Staubli VAL3: testAssembly.dtx

public dio dDio_Sucker = {link=valve1}
public dio dDio_Gripper = {link=valve2}
public tool tTool_3 = {z=179.5, fatherId=flange[0], ioLink=valve2}
public tool tTool_1 = {y=56.52, z=186.17, fatherId=flange[0], ioLink=valve1}
public tool tTool_2 = {y=100, z=136, fatherId=flange[0], ioLink=valve1}
mdesc mNomSpeed
public mdesc mMdesc_Move = {accel=50, vel=50, decel=50, tmax=50000, rmax=50000, leave=25, reach=25}
public mdesc mMdesc_Approach = {accel=20, vel=20, decel=20, tmax=20000, rmax=20000, leave=10, reach=10}
public mdesc mMdesc_Assembly = {accel=10, vel=10, decel=10, tmax=9999, rmax=9999, leave=5, reach=5}
public pointRx pPointRx_Task1[11]
  [0] = {fatherId=world[0]}
  [1] = {x=470.553007, y=-36.92597, z=-100.00047708, rx=-0.00159897, ry=179.996228, rz=0.00184176, fatherId=world[0]}
  [2] = {x=462.557886, y=-40.775959, z=-370.000522428, rx=-0.00112655, ry=179.996342, rz=0.0015039, fatherId=world[0]}
  [3] = {x=462.557886, y=-40.775959, z=-384.955213, rx=-0.00112655, ry=179.996342, rz=0.0015039, fatherId=world[0]}
  [4] = {x=462.557886, y=-40.775959, z=-370.000522428, rx=-0.00112655, ry=179.996342, rz=0.0015039, fatherId=world[0]}
  [5] = {x=462.559535, y=-40.775006, z=-100.00282324, rx=-0.00122429, ry=179.994784, rz=0.00157067, fatherId=world[0]}
  [6] = {x=758.545046, y=166.813373, z=-100.00327697, rx=-0.000742721, ry=179.994769, rz=0.00146888, fatherId=world[0]}
  [7] = {x=755.514304, y=158.963123, z=-333.864783, rx=-0.00147681, ry=179.996751, rz=0.00159201, fatherId=world[0]}
  [8] = {x=755.969382, y=158.33069, z=-366.778404, rx=-0.0014733, ry=179.996625, rz=0.00163886, fatherId=world[0]}
  [9] = {x=755.514304, y=158.963123, z=-333.864783, rx=-0.00147681, ry=179.996751, rz=0.00159201, fatherId=world[0]}
  [10] = {x=755.969382, y=158.33069, z=-100.000545775, rx=-0.00128229, ry=179.995583, rz=0.00173611, fatherId=world[0]}
public pointRx pPointRx_Task2[79]
  [0] = {fatherId=world[0]}
  [1] = {x=784.49936, y=235.445502, z=-49.999237, rx=-2.0204801, ry=113.232882, rz=-88.159509, fatherId=world[0]}
  [2] = {x=786.480486, y=262.552374, z=-299.99927, rx=-2.021757, ry=113.233517, rz=-88.158554, fatherId=world[0]}
  [3] = {x=784.36757, y=256.364439, z=-345.556165, rx=-2.0209842, ry=113.233476, rz=-88.159084, fatherId=world[0]}
  [4] = {x=784.367581, y=247.925511, z=-345.556163, rx=-2.0231337, ry=113.233887, rz=-88.157391, fatherId=world[0]}
  [5] = {x=784.367567, y=246.0220172, z=-341.350417, rx=-2.0233352, ry=113.233862, rz=-88.157219, fatherId=world[0]}
  [6] = {x=784.367581, y=242.656369, z=-336.237706, rx=-2.023434, ry=113.233818, rz=-88.157128, fatherId=world[0]}
  [7] = {x=784.367581, y=237.905853, z=-330.769653, rx=-2.023356, ry=113.233757, rz=-88.15718, fatherId=world[0]}
  [8] = {x=784.367581, y=232.925388, z=-325.864693, rx=-2.0234471, ry=113.233755, rz=-88.157103, fatherId=world[0]}
  [9] = {x=784.367581, y=228.681059, z=-321.473257, rx=-2.0234581, ry=113.233761, rz=-88.157095, fatherId=world[0]}
  [10] = {x=784.36758, y=224.624968, z=-318.39244, rx=-2.023448, ry=113.233762, rz=-88.157103, fatherId=world[0]}
  [11] = {x=784.367571, y=220.157122, z=-315.888328, rx=-2.0231771, ry=113.233735, rz=-88.157321, fatherId=world[0]}
  [12] = {x=784.36758, y=215.623373, z=-312.784136, rx=-2.0234496, ry=113.233801, rz=-88.157109, fatherId=world[0]}
  [13] = {x=784.367578, y=187.857141, z=-309.784137, rx=-2.0235808, ry=113.233878, rz=-88.157017, fatherId=world[0]}
  [14] = {x=784.368404, y=149.380411, z=-325.728255, rx=-2.0259223, ry=113.23421, rz=-88.155082, fatherId=world[0]}
  [15] = {x=784.36842, y=116.303705, z=-343.9057, rx=-2.0259843, ry=113.234309, rz=-88.155037, fatherId=world[0]}
  [16] = {x=786.563391, y=116.321118, z=-358.0200991, rx=-2.0241413, ry=113.234116, rz=-88.156874, fatherId=world[0]}
  [17] = {x=786.563381, y=124.191183, z=-358.108912, rx=-2.0225404, ry=113.233983, rz=-88.158152, fatherId=world[0]}
  [18] = {x=786.563391, y=124.767216, z=-356.140228, rx=-2.0223811, ry=113.233934, rz=-88.158276, fatherId=world[0]}
  [19] = {x=786.563381, y=126.602377, z=-350.283386, rx=-2.0218675, ry=113.233782, rz=-88.158676, fatherId=world[0]}
  [20] = {x=786.563381, y=128.973279, z=-344.998769, rx=-2.021688, ry=113.233689, rz=-88.158812, fatherId=world[0]}
  [21] = {x=786.563381, y=130.903655, z=-341.475635, rx=-2.0216225, ry=113.233645, rz=-88.158861, fatherId=world[0]}
  [22] = {x=786.56339, y=133.536756, z=-336.64486, rx=-2.0217804, ry=113.233636, rz=-88.158733, fatherId=world[0]}
  [23] = {x=786.563381, y=136.419075, z=-333.330297, rx=-2.0221318, ry=113.233692, rz=-88.158455, fatherId=world[0]}
  [24] = {x=786.56338, y=139.330018, z=-329.891057, rx=-2.021782, ry=113.233625, rz=-88.158731, fatherId=world[0]}
  [25] = {x=786.56338, y=143.199956, z=-325.866072, rx=-2.0218296, ry=113.233633, rz=-88.158694, fatherId=world[0]}
  [26] = {x=786.56338, y=146.30778, z=-323.413807, rx=-2.0218444, ry=113.23365, rz=-88.158684, fatherId=world[0]}
  [27] = {x=786.56338, y=149.408417, z=-321.184959, rx=-2.0221042, ry=113.233703, rz=-88.15848, fatherId=world[0]}
  [28] = {x=786.56338, y=154.738391, z=-317.954673, rx=-2.0217603, ry=113.233663, rz=-88.158754, fatherId=world[0]}
  [29] = {x=786.563389, y=158.0830096, z=-315.867788, rx=-2.0216758, ry=113.233652, rz=-88.158821, fatherId=world[0]}
  [30] = {x=786.563379, y=164.0860287, z=-313.649177, rx=-2.0215778, ry=113.233658, rz=-88.158902, fatherId=world[0]}
  [31] = {x=786.563379, y=170.136337, z=-312.205266, rx=-2.0219197, ry=113.233709, rz=-88.158631, fatherId=world[0]}
  [32] = {x=786.563377, y=202.68066, z=-312.205267, rx=-2.0217657, ry=113.233694, rz=-88.158755, fatherId=world[0]}
  [33] = {x=786.562888, y=216.0691273, z=-300.938154, rx=-2.0195136, ry=113.233344, rz=-88.160612, fatherId=world[0]}
  [34] = {x=786.562876, y=231.0113823, z=-300.938159, rx=-2.0171914, ry=113.232942, rz=-88.162452, fatherId=world[0]}
  [35] = {x=786.563361, y=231.0085614, z=-320.286213, rx=-2.0186299, ry=113.233599, rz=-88.161422, fatherId=world[0]}
  [36] = {x=784.474315, y=225.309214, z=-319.0657028, rx=-1.651499, ry=118.747777, rz=-88.567983, fatherId=world[0]}
  [37] = {x=784.474296, y=222.251329, z=-316.987746, rx=-1.652221, ry=118.747936, rz=-88.567442, fatherId=world[0]}
  [38] = {x=784.474315, y=217.578441, z=-314.772279, rx=-1.653461, ry=118.748225, rz=-88.566518, fatherId=world[0]}
  [39] = {x=784.474315, y=215.091758, z=-313.46553, rx=-1.654105, ry=118.748369, rz=-88.566037, fatherId=world[0]}
  [40] = {x=784.474314, y=206.499598, z=-313.465531, rx=-1.654999, ry=118.748116, rz=-88.565412, fatherId=world[0]}
  [41] = {x=784.474089, y=192.932163, z=-313.465215, rx=-1.654882, ry=118.747943, rz=-88.565623, fatherId=world[0]}
  [42] = {x=784.474673, y=178.17243, z=-313.464776, rx=-1.656821, ry=118.748298, rz=-88.564166, fatherId=world[0]}
  [43] = {x=784.474672, y=174.260972, z=-313.464777, rx=-1.656939, ry=118.748314, rz=-88.564078, fatherId=world[0]}
  [44] = {x=784.475657, y=168.377273, z=-315.634673, rx=-1.658494, ry=118.748564, rz=-88.563064, fatherId=world[0]}
  [45] = {x=784.475669, y=164.260614, z=-317.844146, rx=-1.658331, ry=118.748528, rz=-88.563185, fatherId=world[0]}
  [46] = {x=784.475656, y=160.796344, z=-320.542356, rx=-1.658243, ry=118.748527, rz=-88.563255, fatherId=world[0]}
  [47] = {x=784.475656, y=158.320085, z=-323.932867, rx=-1.6584, ry=118.74857, rz=-88.56314, fatherId=world[0]}
  [48] = {x=784.975647, y=155.528626, z=-326.455306, rx=-1.658273, ry=118.748538, rz=-88.563234, fatherId=world[0]}
  [49] = {x=784.976148, y=153.315191, z=-328.0961238, rx=-1.598646, ry=119.905815, rz=-88.631144, fatherId=world[0]}
  [50] = {x=785.626772, y=149.240023, z=-328.814604, rx=-1.599447, ry=120.005925, rz=-88.630678, fatherId=world[0]}
  [51] = {x=786.767462, y=147.46738, z=-331.0758995, rx=-1.60019, ry=120.205812, rz=-88.629945, fatherId=world[0]}
  [52] = {x=787.815814, y=145.632313, z=-333.126809, rx=-1.600796, ry=120.405903, rz=-88.629498, fatherId=world[0]}
  [53] = {x=789.569891, y=142.636972, z=-335.419631, rx=-1.601401, ry=120.555967, rz=-88.629047, fatherId=world[0]}
  [54] = {x=790.459284, y=141.85958, z=-337.809684, rx=-1.559394, ry=120.763388, rz=-88.67702, fatherId=world[0]}
  [55] = {x=791.982542, y=140.32981, z=-341.122996, rx=-1.544512, ry=121.0929413, rz=-88.694365, fatherId=world[0]}
  [56] = {x=792.275209, y=138.662447, z=-342.192906, rx=-1.519234, ry=121.653145, rz=-88.723629, fatherId=world[0]}
  [57] = {x=792.536625, y=138.572731, z=-345.0027193, rx=-1.519371, ry=121.653161, rz=-88.72353, fatherId=world[0]}
  [58] = {x=793.732094, y=138.572712, z=-347.743766, rx=-1.519449, ry=121.653157, rz=-88.723472, fatherId=world[0]}
  [59] = {x=794.288171, y=138.57273, z=-351.481062, rx=-1.519558, ry=121.653153, rz=-88.723392, fatherId=world[0]}
  [60] = {x=795.749739, y=138.572695, z=-352.856774, rx=-1.464073, ry=122.955659, rz=-88.788175, fatherId=world[0]}
  [61] = {x=794.971485, y=136.0698573, z=-356.118195, rx=-1.465483, ry=122.955943, rz=-88.787448, fatherId=world[0]}
  [62] = {x=794.0815342, y=136.0693946, z=-359.869106, rx=-1.418998, ry=124.145823, rz=-88.84234, fatherId=world[0]}
  [63] = {x=793.373601, y=136.0693624, z=-361.302488, rx=-1.441168, ry=123.608884, rz=-88.816781, fatherId=world[0]}
  [64] = {x=792.767182, y=136.0693839, z=-363.47581, rx=-1.441659, ry=123.609108, rz=-88.816452, fatherId=world[0]}
  [65] = {x=792.434025, y=136.0693836, z=-365.777517, rx=-1.441986, ry=123.609244, rz=-88.816232, fatherId=world[0]}
  [66] = {x=792.150715, y=136.0693834, z=-367.211881, rx=-1.442139, ry=123.609301, rz=-88.816129, fatherId=world[0]}
  [67] = {x=791.8949129, y=136.0693916, z=-367.664686, rx=-1.441911, ry=123.609307, rz=-88.816284, fatherId=world[0]}
  [68] = {x=791.881553, y=134.866782, z=-368.123355, rx=-1.442074, ry=123.609311, rz=-88.816161, fatherId=world[0]}
  [69] = {x=791.878458, y=134.86682, z=-369.003385, rx=-1.478326, ry=122.677442, rz=-88.772814, fatherId=world[0]}
  [70] = {x=791.878426, y=134.866796, z=-369.701516, rx=-1.478361, ry=122.677455, rz=-88.77279, fatherId=world[0]}
  [71] = {x=789.693756, y=134.866807, z=-369.700532, rx=-1.478614, ry=122.677609, rz=-88.772623, fatherId=world[0]}
  [72] = {x=787.101896, y=134.866807, z=-369.700532, rx=-1.478507, ry=122.677809, rz=-88.772707, fatherId=world[0]}
  [73] = {x=784.758711, y=134.866807, z=-369.700532, rx=-1.478373, ry=122.677938, rz=-88.772805, fatherId=world[0]}
  [74] = {x=784.162033, y=135.0236018, z=-368.797416, rx=-1.477811, ry=122.677845, rz=-88.773191, fatherId=world[0]}
  [75] = {x=782.666177, y=134.542084, z=-365.000547, rx=-1.477972, ry=122.677921, rz=-88.773082, fatherId=world[0]}
  [76] = {x=782.666175, y=134.542087, z=-350.000824, rx=-1.476616, ry=122.677444, rz=-88.774011, fatherId=world[0]}
  [77] = {x=782.666086, y=134.542023, z=-99.990361, rx=-1.550971, ry=120.912661, rz=-88.686142, fatherId=world[0]}
  [78] = {x=630.68116, y=153.584366, z=-0.0290627, rx=179.85088, ry=-0.0270509, rz=89.981036, fatherId=world[0]}
public pointRx pPointRx_Task3[11]
  [0] = {fatherId=world[0]}
  [1] = {x=457.573791, y=268.618413, z=-93.328799, rx=-0.00378535, ry=-179.998403, rz=89.994828, fatherId=world[0]}
  [2] = {x=453.770842, y=262.862039, z=-349.998607, rx=-0.0391003, ry=-179.998515, rz=88.347078, fatherId=world[0]}
  [3] = {x=453.770842, y=262.862039, z=-370.925588, rx=-0.0392417, ry=-179.998183, rz=88.347077, fatherId=world[0]}
  [4] = {x=453.770842, y=262.862039, z=-349.998607, rx=-0.0391003, ry=-179.998515, rz=88.347078, fatherId=world[0]}
  [5] = {x=453.77274, y=262.862555, z=-93.330348, rx=-0.0381543, ry=-179.999602, rz=88.347097, fatherId=world[0]}
  [6] = {x=822.0424047, y=164.484092, z=-93.329995, rx=-0.03848, ry=-179.999434, rz=88.347127, fatherId=world[0]}
  [7] = {x=820.569687, y=155.795627, z=-319.99874, rx=-0.0379678, ry=-179.997835, rz=88.914173, fatherId=world[0]}
  [8] = {x=820.568927, y=155.794808, z=-351.1718049, rx=-0.0379487, ry=-179.997795, rz=88.914233, fatherId=world[0]}
  [9] = {x=820.56972, y=155.795377, z=-319.99874, rx=-0.038019, ry=-179.997841, rz=88.914331, fatherId=world[0]}
  [10] = {x=820.569682, y=155.795626, z=-93.332919, rx=-0.0378152, ry=-179.998731, rz=88.914356, fatherId=world[0]}
public jointRx jJointRx_Task2[79]
  [1] = {j1=17.0735993, j2=33.71783, j3=87.23164, j4=68.492033, j5=-17.714491, j6=-150.61}
  [2] = {j1=19.267617, j2=57.807089, j3=85.658836, j4=34.598768, j5=-33.858209, j6=-111.939597}
  [3] = {j1=18.819866, j2=62.533953, j3=84.516221, j4=31.17674, j5=-36.73072, j6=-108.199587}
  [4] = {j1=18.121718, j2=62.29358, j3=85.15009, j4=29.88914, j5=-36.877659, j6=-107.324371}
  [5] = {j1=17.963337, j2=61.761476, j3=85.502305, j4=29.776456, j5=-36.679155, j6=-107.350149}
  [6] = {j1=17.682478, j2=61.0872296, j3=85.997367, j4=29.481484, j5=-36.448185, j6=-107.276726}
  [7] = {j1=17.284343, j2=60.223956, j3=86.641455, j4=29.0357207, j5=-36.150959, j6=-107.137831}
  [8] = {j1=16.864874, j2=59.534662, j3=87.211953, j4=28.486656, j5=-35.936335, j6=-106.892884}
  [9] = {j1=16.505728, j2=59.0386009, j3=87.652003, j4=27.982906, j5=-35.793746, j6=-106.64176}
  [10] = {j1=16.161093, j2=58.58449, j3=88.0572361, j4=27.493562, j5=-35.662339, j6=-106.393662}
  [11] = {j1=15.779851, j2=58.186535, j3=88.457586, j4=26.91314, j5=-35.56863, j6=-106.0714424}
  [12] = {j1=15.391393, j2=57.94679, j3=88.796721, j4=26.259704, j5=-35.562015, j6=-105.667212}
  [13] = {j1=12.9768, j2=57.296772, j3=90.461477, j4=21.997304, j5=-35.954017, j6=-102.91758}
  [14] = {j1=9.539802, j2=57.822964, j3=91.923306, j4=15.919761, j5=-37.254771, j6=-99.00833214}
  [15] = {j1=6.513776, j2=59.485822, j3=92.372855, j4=10.823729, j5=-38.968332, j6=-95.890175}
  [16] = {j1=6.492073, j2=61.306077, j3=91.23944, j4=10.635004, j5=-39.641375, j6=-95.671847}
  [17] = {j1=7.214447, j2=61.414554, j3=90.951075, j4=11.713001, j5=-39.529681, j6=-96.239868}
  [18] = {j1=7.267197, j2=61.186984, j3=91.0371749, j4=11.823806, j5=-39.396227, j6=-96.322933}
  [19] = {j1=7.435141, j2=60.513766, j3=91.280904, j4=12.175813, j5=-38.992631, j6=-96.585887}
  [20] = {j1=7.651943, j2=59.919078, j3=91.46309, j4=12.601734, j5=-38.611947, j6=-96.887767}
  [21] = {j1=7.828264, j2=59.529423, j3=91.565028, j4=12.940354, j5=-38.350141, j6=-97.122896}
  [22] = {j1=8.0685012, j2=58.997817, j3=91.697139, j4=13.41095, j5=-37.987817, j6=-97.454453}
  [23] = {j1=8.331086, j2=58.651028, j3=91.738585, j4=13.894013, j5=-37.721548, j6=-97.776617}
  [24] = {j1=8.595708, j2=58.292528, j3=91.778761, j4=14.390068, j5=-37.445015, j6=-98.11279}
  [25] = {j1=8.946867, j2=57.88365, j3=91.798001, j4=15.0478112, j5=-37.112936, j6=-98.557681}
  [26] = {j1=9.228256, j2=57.648841, j3=91.772361, j4=15.564104, j5=-36.899352, j6=-98.90043}
  [27] = {j1=9.508476, j2=57.441955, j3=91.732612, j4=16.0791221, j5=-36.701035, j6=-99.242661}
  [28] = {j1=9.988714, j2=57.160428, j3=91.628813, j4=16.958271, j5=-36.401989, j6=-99.824779}
  [29] = {j1=10.289208, j2=56.979718, j3=91.560199, j4=17.518577, j5=-36.210178, j6=-100.201582}
  [30] = {j1=10.826799, j2=56.835937, j3=91.363344, j4=18.48848, j5=-35.973345, j6=-100.83541}
  [31] = {j1=11.366347, j2=56.787405, j3=91.120709, j4=19.450609, j5=-35.790773, j6=-101.457762}
  [32] = {j1=14.224669, j2=57.4931, j3=89.316, j4=24.431809, j5=-35.347537, j6=-104.622003}
  [33] = {j1=15.377286, j2=56.563894, j3=88.918111, j4=27.0434156, j5=-34.430933, j6=-106.639166}
  [34] = {j1=16.64669, j2=56.96649, j3=87.92593, j4=29.426616, j5=-34.254434, j6=-108.263593}
  [35] = {j1=16.646633, j2=59.120348, j3=87.153514, j4=28.467866, j5=-35.462896, j6=-107.0950929}
  [36] = {j1=15.767302, j2=58.243823, j3=85.248349, j4=32.882189, j5=-27.605831, j6=-112.0659061}
  [37] = {j1=15.513217, j2=57.933793, j3=85.529788, j4=32.464444, j5=-27.500121, j6=-111.824926}
  [38] = {j1=15.123585, j2=57.566476, j3=85.917056, j4=31.75416, j5=-27.393722, j6=-111.377185}
  [39] = {j1=14.915571, j2=57.35816, j3=86.124365, j4=31.384947, j5=-27.328046, j6=-111.149607}
  [40] = {j1=14.193118, j2=57.134808, j3=86.664735, j4=29.779347, j5=-27.383454, j6=-109.996923}
  [41] = {j1=13.0412292, j2=56.801837, j3=87.47303, j4=27.264233, j5=-27.478278, j6=-108.213867}
  [42] = {j1=11.774113, j2=56.466939, j3=88.289523, j4=24.561833, j5=-27.58992, j6=-106.329643}
  [43] = {j1=11.435863, j2=56.38286, j3=88.49517, j4=23.850233, j5=-27.620891, j6=-105.838586}
  [44] = {j1=10.925508, j2=56.500278, j3=88.717436, j4=22.667109, j5=-27.817494, j6=-104.974556}
  [45] = {j1=10.566933, j2=56.662581, j3=88.840859, j4=21.811619, j5=-28.00483888, j6=-104.340331}
  [46] = {j1=10.264405, j2=56.895235, j3=88.907969, j4=21.0593036, j5=-28.221481, j6=-103.77059}
  [47] = {j1=10.0477658, j2=57.226862, j3=88.895701, j4=20.460011, j5=-28.477105, j6=-103.293598}
  [48] = {j1=9.803071, j2=57.457636, j3=88.92735, j4=19.856107, j5=-28.676626, j6=-102.83763}
  [49] = {j1=9.547973, j2=57.545403, j3=88.337249, j4=20.279081, j5=-27.0284365, j6=-103.432976}
  [50] = {j1=9.17554, j2=57.636815, j3=88.28089, j4=19.563048, j5=-26.990242, j6=-102.975457}
  [51] = {j1=9.00483014, j2=57.942233, j3=88.0585164, j4=19.191456, j5=-27.037077, j6=-102.716881}
  [52] = {j1=8.830323, j2=58.216856, j3=87.861525, j4=18.817473, j5=-27.0787177, j6=-102.459381}
  [53] = {j1=8.545627, j2=58.551375, j3=87.570421, j4=18.260321, j5=-27.0694017, j6=-102.0989601}
  [54] = {j1=8.426197, j2=58.842246, j3=86.85934, j4=18.711904, j5=-25.81163, j6=-102.634657}
  [55] = {j1=8.259178, j2=59.291415, j3=86.311308, j4=18.620537, j5=-25.366142, j6=-102.656307}
  [56] = {j1=8.0591997, j2=59.560727, j3=85.541231, j4=18.866688, j5=-24.308967, j6=-103.0590384}
  [57] = {j1=8.0386162, j2=59.951453, j3=85.222676, j4=18.773893, j5=-24.373487, j6=-102.975711}
  [58] = {j1=8.0241566, j2=60.346473, j3=84.87483, j4=18.711457, j5=-24.415521, j6=-102.920183}
  [59] = {j1=8.00541723, j2=60.879947, j3=84.409807, j4=18.625734, j5=-24.47697, j6=-102.842921}
  [60] = {j1=7.942356, j2=61.0649335, j3=83.487014, j4=19.811859, j5=-22.500867, j6=-104.07919}
  [61] = {j1=7.727508, j2=61.401843, j3=83.399621, j4=19.157352, j5=-22.694586, j6=-103.560246}
  [62] = {j1=7.709323, j2=61.611067, j3=83.0617261, j4=19.986652, j5=-21.414562, j6=-104.371287}
  [63] = {j1=7.750401, j2=61.647608, j3=83.614499, j4=19.241429, j5=-22.499143, j6=-103.576108}
  [64] = {j1=7.772676, j2=61.746555, j3=83.878384, j4=19.00464446, j5=-22.845946, j6=-103.299559}
  [65] = {j1=7.782473, j2=61.942167, j3=83.927587, j4=18.838225, j5=-23.079234, j6=-103.109987}
  [66] = {j1=7.784648, j2=62.0896024, j3=83.89288, j4=18.757943, j5=-23.186307, j6=-103.02071}
  [67] = {j1=7.791107, j2=62.20162, j3=83.932528, j4=18.657764, j5=-23.33108, j6=-102.905854}
  [68] = {j1=7.679016, j2=62.37023, j3=83.773947, j4=18.420191, j5=-23.32075, j6=-102.748476}
  [69] = {j1=7.719182, j2=62.55715, j3=84.240192, j4=17.56371, j5=-24.859608, j6=-101.849277}
  [70] = {j1=7.719188, j2=62.613636, j3=84.214779, j4=17.543559, j5=-24.889227, j6=-101.827056}
  [71] = {j1=7.7448, j2=62.45529, j3=84.630459, j4=17.428262, j5=-25.138746, j6=-101.676102}
  [72] = {j1=7.775314, j2=62.269126, j3=85.121259, j4=17.29483, j5=-25.434224, j6=-101.50015}
  [73] = {j1=7.8031, j2=62.102288, j3=85.562859, j4=17.177779, j5=-25.700925, j6=-101.344414}
  [74] = {j1=7.823739, j2=61.799348, j3=85.785297, j4=17.266053, j5=-25.627329, j6=-101.423074}
  [75] = {j1=7.799701, j2=61.454504, j3=86.186419, j4=17.185676, j5=-25.677214, j6=-101.356406}
  [76] = {j1=7.799425, j2=59.474328, j3=87.00387612, j4=17.931263, j5=-24.568895, j6=-102.180284}
  [77] = {j1=7.87704, j2=35.0821518, j3=89.427363, j4=66.459413, j5=-8.237557, j6=-152.186423}
  [78] = {j1=8.0787279, j2=40.991134, j3=60.528262, j4=-0.14677, j5=78.528442, j6=-81.910768}
public jointRx jJointRx_Task3[11]
  [1] = {j1=25.00925885, j2=15.870786, j3=105.718793, j4=-0.0032346, j5=58.413468, j6=115.00578125}
  [2] = {j1=24.630506, j2=42.659059, j3=111.667536, j4=-0.0805587, j5=25.691073, j6=113.0501848}
  [3] = {j1=24.6305, j2=45.414499, j3=111.0900932, j4=-0.0875116, j5=23.513438, j6=113.0578287}
  [4] = {j1=24.630506, j2=42.659059, j3=111.667536, j4=-0.0805587, j5=25.691073, j6=113.0501848}
  [5] = {j1=24.630252, j2=15.138536, j3=106.681375, j4=-0.0406148, j5=58.196359, j6=112.998759}
  [6] = {j1=7.908445, j2=58.734796, j3=35.90856, j4=-0.0381611, j5=85.3625, j6=96.25866}
  [7] = {j1=7.330912, j2=70.374183, j3=45.167482, j4=-0.0414276, j5=64.465455, j6=96.262946}
  [8] = {j1=7.330854, j2=72.937204, j3=44.415778, j4=-0.0421143, j5=62.654053, j6=96.26441}
  [9] = {j1=7.330912, j2=70.374183, j3=45.167482, j4=-0.0414276, j5=64.465334, j6=96.262946}
  [10] = {j1=7.330899, j2=58.0329479, j3=37.210714, j4=-0.0375007, j5=84.762424, j6=96.24868}
public jointRx jJointRx_Task1[11]
  [1] = {j1=-17.2143, j2=9.687656, j3=113.521032, j4=-0.00049125, j5=56.787236, j6=-17.212189}
  [2] = {j1=-17.950805, j2=41.543882, j3=119.486958, j4=0.000171665, j5=18.965332, j6=-17.949463}
  [3] = {j1=-17.950805, j2=43.710476, j3=118.997734, j4=0.000187737, j5=17.287962, j6=-17.94948}
  [4] = {j1=-17.950805, j2=41.543882, j3=119.486958, j4=0.000171665, j5=18.965332, j6=-17.949463}
  [5] = {j1=-17.950871, j2=8.810998, j3=114.566701, j4=0.0005305, j5=56.616962, j6=-17.949592}
  [6] = {j1=4.533296, j2=45.753264, j3=59.299507, j4=-0.00119486, j5=74.942073, j6=4.535076}
  [7] = {j1=3.962357, j2=60.776818, j3=66.124055, j4=-0.00212317, j5=53.0959886, j6=3.965223}
  [8] = {j1=3.912499, j2=63.798827, j3=65.304217, j4=-0.00219096, j5=50.893689, j6=3.91552}
  [9] = {j1=3.962357, j2=60.776818, j3=66.124055, j4=-0.00212317, j5=53.0959886, j6=3.965223}
  [10] = {j1=3.912455, j2=45.191575, j3=60.27581, j4=-0.00164014, j5=74.528296, j6=3.914629}
public tool tTool_flange = {fatherId=flange[0], ioLink=valve1}
public jointRx jJointRx_Asse_E = {j1=-0.0013705, j2=22.326988, j3=78.0153817, j4=-0.000755365, j5=79.653327, j6=0.000168207}
public pointRx pPointRx_Asse_S = {x=629.572969, y=106.501229, z=30.667254, rx=-0.000743185, ry=179.995697, rz=0.0014031, fatherId=world[0]}
public pointRx pPointRx_Asse_E = {x=629.572969, y=106.501229, z=30.667254, rx=-0.000743185, ry=179.995697, rz=0.0014031, fatherId=world[0]}
public jointRx jJointRx_Asse_S = {j1=-0.0013705, j2=22.326988, j3=78.0153817, j4=-0.000755365, j5=79.653327, j6=0.000168207}
public jointRx jJointRx_Init
